{attribute 'linkalways'} 
{attribute 'no_explicit_call' := 'This FB is a CLASS and must be accessed using methods or properties'}
{attribute 'enable_dynamic_creation'}
FUNCTION_BLOCK BuildXYZGroupCommand EXTENDS NciCommand
VAR
	_fb : CfgBuild3DGroup;
	_groupId : UDINT;
	_xAxisId : UDINT;
	_yAxisId : UDINT;
	_zAxisId : UDINT;
	_timeout : TIME;
END_VAR

METHOD FB_init : BOOL
VAR_INPUT
	bInitRetains : BOOL; // if TRUE, the retain variables are initialized (warm start / cold start)
	bInCopyCode : BOOL;  // if TRUE, the instance afterwards gets moved into the copy code (online change)
	nci : I_Nci := 0;
	xAxis : I_Axis := 0;
	yAxis : I_Axis := 0;
	zAxis : I_Axis := 0;
	timeout : TIME;
END_VAR
_groupId := nci.GroupId;
IF xAxis <> 0 THEN
	_xAxisId := xAxis.AxisId;
END_IF
IF yAxis <> 0 THEN
	_yAxisId := yAxis.AxisId;
END_IF
IF zAxis <> 0 THEN
	_zAxisId := zAxis.AxisId;
END_IF
_timeout := timeout;
END_METHOD

METHOD PROTECTED  WhileBusy
VAR_INPUT
	CommandState : I_CommandBusyState;
END_VAR
_fb(
	bExecute := TRUE,
	nGroupId := _groupId,
	nXAxisId := _xAxisId,
	nYAxisId := _yAxisId,
	nZAxisId := _zAxisId,
	tTimeOut := _timeout,
);

IF _fb.bBusy THEN
	RETURN;
END_IF

IF _fb.bErr THEN
	CommandState.SetError(_fb.nErrId);
	_fb(bExecute := FALSE);
	RETURN;
END_IF

_fb(bExecute := FALSE);
CommandState.SetDone();
END_METHOD

END_FUNCTION_BLOCK

(* stored: Version 1.1.0.1, ProductVersion 3.1.4024.12
   POU BuildXYZGroupCommand: Id {1ff9de8f-fa12-49cf-bac9-4763061f268a}, SpecialFunc None
   Method FB_init: Id {4cede08a-9c65-433d-b392-038dd509d411}
   Method WhileBusy: Id {da1a010e-4772-4e0b-a2f6-e72690e4d72e} *)
